FUNCTION_BLOCK FB_HomeDS402 IMPLEMENTS I_HomeDS402
VAR_INPUT
END_VAR
VAR_OUTPUT
END_VAR
VAR
    iMotionLogger : I_MotionLogger;
    //iLimSwStatus : I_LimSwStatus;
    //iHomeShareData : I_HomeShareData ;
    bCommandMoveHome  : BOOL;
    bBusy	: BOOL;
    bDone	: BOOL;
    bError 	: BOOL;
    bAbort   : BOOL;
    bAborted  : BOOL;
    nErrorID : UDINT;
    fOffset  : LREAL;
    fPosition	: LREAL;
    rtDone	: R_TRIG;
    fHomeSpeedFast	: LREAL;
    fHomeSpeedSlow	: LREAL;
    bBit13OpModeSpecific	: BOOL;
    bBit12OpModeSpecific	: BOOL;
    bTargetReached	: BOOL;
    nDriveControl : UINT;
    nModeOfOperation : SINT;
    nModeOfOperationDisplay : SINT;
    nMostRecentModeOfOperation : SINT;
    eHomeMode: E_EpicsHomeCmd :=E_EpicsHomeCmd.AUTOZERO;
    rtExec: R_TRIG;
    ftExec: F_TRIG;
    bMove  : BOOL;
    tonSyncHoming : TON;
    {attribute 'hide'}
    eHomeState	: E_MoveState;
    rtReset: R_TRIG;
    bReset: BOOL;
    sMessage: T_MAXSTRING;
END_VAR

//NB: The calling must pass drive status register.
THIS^.rtExec(CLK:=THIS^.bCommandMoveHome);
THIS^.ftExec(CLK:=THIS^.bCommandMoveHome);

tonSyncHoming(PT:=T#50MS);
CASE THIS^.eHomeMode OF
    E_EpicsHomeCmd.AUTOZERO:
        THIS^.bMove := TRUE;
    E_EpicsHomeCmd.NONE:
        THIS^.bMove := FALSE;
        THIS^.bBusy := THIS^.rtExec.Q;
        THIS^.bDone := NOT THIS^.rtExec.Q;
    ELSE
        THIS^.bMove := FALSE;
END_CASE

IF THIS^.bMove THEN
    IF THIS^.bBusy AND THIS^.ftExec.Q THEN
        THIS^.eHomeState := E_MoveState.ERROR;
        THIS^.bAborted := TRUE;
    END_IF
    CASE eHomeState OF
        // Wait for a rising edge
        E_MoveState.IDLING:
            IF THIS^.rtExec.Q THEN
                THIS^.bDone := FALSE;
                THIS^.bBusy := TRUE;
                THIS^.bError := FALSE;
                THIS^.nErrorID := 0;
                THIS^.bAborted := FALSE;
                THIS^.eHomeState := E_MoveState.INIT;
                // make sure the run flag is clear, this would be the case
                // in EnableMode ->ALWAYS and ModeofOperation ->CSP
                nDriveControl:=15;
                THIS^.tonSyncHoming.IN := TRUE;
            END_IF
        E_MoveState.INIT:
            // sdo write homing paramters;
            // This mode will be restore after homing
            THIS^.nMostRecentModeOfOperation := nModeOfOperationDisplay;
            nDriveControl:=31;
            // take some time for drive to register above commad and start
            // homming routine.
            IF tonSyncHoming.Q THEN
              eHomeState:=E_MoveState.STARTED;
            END_IF

        E_MoveState.STARTED :
            // this is a comfirmation that routine is ongoing
            IF NOT bTargetReached
               AND NOT bBit13OpModeSpecific THEN
                bBusy:=TRUE;
                bDone:=FALSE;
                eHomeState:=E_MoveState.IN_PROGRESS;
            END_IF
        E_MoveState.IN_PROGRESS :
            // Genral Motion error i.e Following error ?
            IF bBit13OpModeSpecific THEN
                eHomeState:=E_MoveState.ERROR;
            // Reached
            ELSIF bTargetReached
                AND bBit12OpModeSpecific
                AND NOT bBit13OpModeSpecific THEN
                eHomeState:=E_MoveState.REACHED;
            END_IF

        E_MoveState.REACHED:
            bBusy:=FALSE;
            bDone:=TRUE;
            //prepare next move
            nDriveControl:=15;
            // Restore default mode
            nModeOfOperation:=THIS^.nMostRecentModeOfOperation;
            tonSyncHoming.IN := FALSE;
        E_MoveState.ERROR:
            bError:= TRUE;
            bDone:=FALSE;
            // sdo read in case of error
            // HomeErrorID
            bBusy:= FALSE;
    END_CASE
END_IF

//NB: The calling must forward control register for i/o update.
// Reset execute after when done successfull or after abort reset
// this way the done and error condition is latched till next move or global reset.
rtDone(CLK:=bDone);
IF  rtDone.Q  THEN
    THIS^.bCommandMoveHome := FALSE;
END_IF

// an interruption can be external i.e, an halt, Reset or a local condition
THIS^.rtReset(CLK:=bReset);
IF THIS^.rtReset.Q THEN
    THIS^.bError := FALSE;
    THIS^.nErrorID := 0;
    THIS^.bAborted := FALSE;
    THIS^.sMessage := '';
	THIS^.bReset := FALSE;
END_IF

PROPERTY Aborted : BOOL
GET
Aborted := bAborted;
END_GET
END_PROPERTY

{warning 'Add property implementation'}
PROPERTY Active : BOOL
GET
END_GET
END_PROPERTY

{warning 'add property implementation'}
PROPERTY Busy : BOOL
GET
Busy := THIS^.bBusy;
END_GET
END_PROPERTY

METHOD PUBLIC CallAfterInit
VAR_INPUT
    iMotionLogger : I_MotionLogger;
END_VAR
THIS^.iMotionLogger := iMotionLogger;
END_METHOD

{warning 'Add property implementation'}
PROPERTY CommandMoveHome : BOOL
SET
bCommandMoveHome := CommandMoveHome;
END_SET
END_PROPERTY

{warning 'add property implementation'}
PROPERTY Done : BOOL
GET
Done := THIS^.bDone;
END_GET
END_PROPERTY

PROPERTY DS402Control : UINT
GET
DS402Control := nDriveControl;
END_GET
END_PROPERTY

PROPERTY DS402ModeOfOperation : SINT
GET
DS402ModeOfOperation  := nModeOfOperation;
END_GET
END_PROPERTY

METHOD DS402Status
VAR_INPUT
    ModeOfOperationDisplay : SINT;
    Bit13OpModeSpecific	: BOOL;
    Bit12OpModeSpecific	: BOOL;
    TargetReached	: BOOL;
END_VAR
nModeOfOperationDisplay := ModeOfOperationDisplay;
bBit13OpModeSpecific := Bit13OpModeSpecific;
bBit12OpModeSpecific := Bit12OpModeSpecific;
bTargetReached := TargetReached;
END_METHOD

{warning 'add property implementation'}
PROPERTY Error : BOOL
GET
Error := THIS^.bError;
END_GET
END_PROPERTY

{warning 'add property implementation'}
PROPERTY ErrorID : UDINT
GET
ErrorID := THIS^.nErrorID;
END_GET
END_PROPERTY

//FB_Init is always available implicitly and it is used primarily for initialization.
//The return value is not evaluated. For a specific influence, you can also declare the
//methods explicitly and provide additional code there with the standard initialization
//code. You can evaluate the return value.
METHOD FB_Init: BOOL
VAR_INPUT
    bInitRetains: BOOL; // TRUE: the retain variables are initialized (reset warm / reset cold)
    bInCopyCode: BOOL;  // TRUE: the instance will be copied to the copy code afterward (online change)
    iMotionLogger : I_MotionLogger;
END_VAR
THIS^.iMotionLogger := iMotionLogger;
END_METHOD

{warning 'Add property implementation'}
PROPERTY GlobalReset : BOOL
SET
bReset := GlobalReset;
END_SET
END_PROPERTY

METHOD Home
VAR_INPUT
    Execute	: BOOL;
    HomeSpeedFast	: LREAL;
    HomeSpeedSlow	: LREAL;
END_VAR
THIS^.bCommandMoveHome := Execute;
THIS^.fHomeSpeedFast := HomeSpeedFast;
THIS^.fHomeSpeedSlow := HomeSpeedSlow;
END_METHOD

PROPERTY Message : T_MAXSTRING
GET
Message := sMessage;
END_GET
END_PROPERTY

PROPERTY Mode : E_EpicsHomeCmd
GET
Mode := eHomeMode;
END_GET
SET
eHomeMode := Mode;
END_SET
END_PROPERTY

{warning 'Add property implementation'}
PROPERTY Offset : LREAL
SET
fOffset := Offset;
END_SET
END_PROPERTY

{warning 'Add property implementation'}
PROPERTY Position : LREAL
SET
fPosition := Position;
END_SET
END_PROPERTY

END_FUNCTION_BLOCK

(* stored: Version 1.1.0.1
   POU FB_HomeDS402: Id {fbf9953c-abc4-4ff2-b40d-41861c6228fc}, SpecialFunc None
   Property Aborted: Id {f628076d-da64-46a3-9b2e-51ef77ba2849}
   Get Get: Id {f866410a-aefc-4817-8d05-a7966bf27315}
   Property Active: Id {2ec4b934-b83b-40a1-89e4-42fd9450a9e9}
   Get Get: Id {5ce1d2b4-0255-47fe-9b81-ea8d68a1187a}
   Property Busy: Id {08f4c53a-a93f-4c0f-81a4-fc4b91c13ab5}
   Get Get: Id {a9f0aa36-9754-42d8-8ac1-0e120c0daa7f}
   Method CallAfterInit: Id {fe9db625-490b-485d-a2d4-bb34c240c290}
   Property CommandMoveHome: Id {ee03e6b2-d0a1-4de6-8b3b-367209048f73}
   Set Set: Id {b98b121c-ddb6-47db-8c64-61500ddff177}
   Property Done: Id {4f9baf15-b527-487e-8710-a14003009a1c}
   Get Get: Id {0b073f86-ebf7-4ab3-9e80-887fc0329919}
   Property DS402Control: Id {4033051e-3bcc-421f-84e9-2fa7f78a1b85}
   Get Get: Id {6da058be-1b97-4f09-8c0f-91efc034b490}
   Property DS402ModeOfOperation: Id {5f3be5b6-0454-423f-adb3-6186fe16b30b}
   Get Get: Id {aa592275-3499-4171-9be7-f81686ae87bb}
   Method DS402Status: Id {d99216d5-05a0-4090-ab57-79a7bde36202}
   Property Error: Id {032eb170-b5c9-4f58-baf7-a259d7549383}
   Get Get: Id {1fdeb09e-0529-4586-8f44-e19b71367709}
   Property ErrorID: Id {d931b1ca-ae52-4471-a302-e9584e38504b}
   Get Get: Id {2d6153ac-27f4-46d6-a224-787a0075982c}
   Method FB_Init: Id {8f57f631-0cc5-486a-b712-0c732bc45c46}
   Property GlobalReset: Id {8a55c20f-6ca9-433d-9fd5-e4475bd1b3c1}
   Set Set: Id {1d005cd5-1cf0-4011-b545-7f7f15def153}
   Method Home: Id {e9200b22-57ed-4146-80d4-2882e00b73f4}
   Property Message: Id {8a09e656-584e-42d0-b55b-a832eece117d}
   Get Get: Id {ad47af60-da43-4f64-8c36-cc22f2c3972a}
   Property Mode: Id {ae75dbc7-8132-452c-bcd4-63471502db3c}
   Get Get: Id {77995d4e-8083-4845-ada0-e17537ce5f9a}
   Set Set: Id {eb23e651-ed2b-47ef-a422-ccd55362cca4}
   Property Offset: Id {8c816e30-0a55-412d-a75b-c41529942f5a}
   Set Set: Id {d4b4ef7f-b15c-44ed-8ced-865f552cbcaa}
   Property Position: Id {1a510ee5-ff47-4454-aa3c-a3b17a57e147}
   Set Set: Id {3dc8b970-b6c7-4d4d-9a14-299692f00a16} *)
